Staubli VAL3: Pionperdu.pgx

program Pionperdu(num x_nPionperdu (dimensions=1), num x_nPionjete (dimensions=1))
begin
  //met à jour position des cases noires

  //Deplacementpion(X,Y) -> deplacement du pion de X vers Y


  //Deplacement vers le pion en X
  movej(appro(pCaseNoire[x_nPionperdu],trAppro),tTool,mDeplacement)

  //s'approche et prend le pion en X
  close(tTool)
  movel(pCaseNoire[x_nPionperdu],tTool,mPrise)
  open(tTool)

  movel(appro(pCaseNoire[x_nPionperdu],trAppro),tTool,mDeplacement)

  //Deplacement vers Y puis approche vers Y
  movej(appro(pPieceMangees[x_nPionjete],trAppro),tTool,mDeplacement)
  movel(pPieceMangees[x_nPionjete],tTool,mPrise)

  //lache la piece et remonte
  close(tTool)
  movel(appro(pPieceMangees[x_nPionjete],trAppro),tTool,mDeplacement)


end
